FUNCTION_BLOCK FB_MadgwickFilter
VAR_INPUT
    stAccelData : ST_3D_values; // Acceleration Data in (g)
    stGyroData : ST_3D_values; // Gyroscope Data in (°/s)
    fBeta: REAL := 0.05; // Algorithm gain
    fCycletime: REAL; // Time step (s)
    bSetReference: BOOL; // Flag to set reference position
END_VAR

VAR_OUTPUT
	fQ0 : LREAL := 1.0; // Quaternion component
    fQ1 : LREAL := 0.0; // Quaternion component
    fQ2 : LREAL := 0.0; // Quaternion component
    fQ3 : LREAL := 0.0; // Quaternion component
    stEulerAngle_deg : ST_3D_values; // Estimated Euler angle in degrees X= Pitch, Y=Roll, Z=Yaw
    stEulerAngle_rad : ST_3D_values; // Estimated Euler angle in rad X= Pitch, Y=Roll, Z=Yaw
END_VAR

VAR

	// Reference angles
	stRef_Angles_deg :ST_3d_values; // Reference orientation (bSetReference; angles in degrees)
    fNorm : LREAL;
    _2fQ0, _2fQ1, _2fQ2, _2fQ3 : LREAL;
    _4fQ0, _4fQ1, _4fQ2, _4fQ3 : LREAL;
    _8fQ1, _8fQ2 : LREAL;
    fQ0fQ0, fQ1fQ1, fQ2fQ2, fQ3fQ3 : LREAL;
    fAx, fAy, fAz : LREAL;
    fS1, fS2, fS3, fS4 : LREAL;
    fSinRoll, fCosRoll : LREAL;
    fSinPitch, fCosPitch : LREAL;
    fSinYaw, fCosYaw : LREAL;
	fGyroRateX_rad,fGyroRateY_rad, fGyroRateZ_rad:LREAL;
END_VAR

// Normalize accelerometer measurements
fAx := REAL_TO_LREAL(stAccelData.x);
fAy := REAL_TO_LREAL(stAccelData.y);
fAz := REAL_TO_LREAL(stAccelData.z);
fNorm := fAx * fAx + fAy * fAy + fAz * fAz;
IF fNorm > 1E-6 THEN
    fNorm := SQRT(fNorm);
    fAx := fAx / fNorm;
    fAy := fAy / fNorm;
    fAz := fAz / fNorm;
END_IF

// Estimated direction of gravity and magnetic field
_2fQ0 := 2.0 * fQ0;
_2fQ1 := 2.0 * fQ1;
_2fQ2 := 2.0 * fQ2;
_2fQ3 := 2.0 * fQ3;
_4fQ0 := 4.0 * fQ0;
_4fQ1 := 4.0 * fQ1;
_4fQ2 := 4.0 * fQ2;
_4fQ3 := 4.0 * fQ3;
_8fQ1 := 8.0 * fQ1;
_8fQ2 := 8.0 * fQ2;
fQ0fQ0 := fQ0 * fQ0;
fQ1fQ1 := fQ1 * fQ1;
fQ2fQ2 := fQ2 * fQ2;
fQ3fQ3 := fQ3 * fQ3;

// Gradient descent algorithm corrective step
fS1 := _4fQ0 * fQ2fQ2 + _2fQ2 * fAx + _4fQ0 * fQ1fQ1 - _2fQ1 * fAy;
fS2 := _4fQ1 * fQ3fQ3 - _2fQ3 * fAx + 4.0 * fQ0fQ0 * fQ1 - _2fQ0 * fAy - _4fQ1 + _8fQ1 * fQ1fQ1 + _8fQ1 * fQ2fQ2 + _4fQ1 * fAz;
fS3 := 4.0 * fQ0fQ0 * fQ2 + _2fQ0 * fAx + _4fQ2 * fQ3fQ3 - _2fQ3 * fAy - _4fQ2 + _8fQ2 * fQ1fQ1 + _8fQ2 * fQ2fQ2 + _4fQ2 * fAz;
fS4 := 4.0 * fQ1fQ1 * fQ3 - _2fQ1 * fAx + 4.0 * fQ2fQ2 * fQ3 - _2fQ2 * fAy;

// Normalize step magnitude
fNorm := fS1 * fS1 + fS2 * fS2 + fS3 * fS3 + fS4 * fS4;
IF fNorm > 1E-6 THEN
    fNorm := SQRT(fNorm);
    fS1 := fS1 / fNorm;
    fS2 := fS2 / fNorm;
    fS3 := fS3 / fNorm;
    fS4 := fS4 / fNorm;
END_IF

// Apply gradient descent corrective step
fQ0 := fQ0 - REAL_TO_LREAL(fBeta) * fS1 * REAL_TO_LREAL(fCycleTime);
fQ1 := fQ1 - REAL_TO_LREAL(fBeta) * fS2 * REAL_TO_LREAL(fCycleTime);
fQ2 := fQ2 - REAL_TO_LREAL(fBeta) * fS3 * REAL_TO_LREAL(fCycleTime);
fQ3 := fQ3 - REAL_TO_LREAL(fBeta) * fS4 * REAL_TO_LREAL(fCycleTime);

// Convert gyroscope rates from °/s to rad/s
fGyroRateX_rad := stGyroData.x * pi / 180.0;
fGyroRateY_rad := stGyroData.y * pi / 180.0;
fGyroRateZ_rad := stGyroData.z * pi / 180.0;

// Integrate rate of change of quaternion
fQ0 := fQ0 + 0.5 * (-fQ1 * REAL_TO_LREAL(fGyroRateX_rad) - fQ2 * REAL_TO_LREAL(fGyroRateY_rad) - fQ3 * REAL_TO_LREAL(fGyroRateZ_rad)) * REAL_TO_LREAL(fCycleTime);
fQ1 := fQ1 + 0.5 * (fQ0 * REAL_TO_LREAL(fGyroRateX_rad) + fQ2 * REAL_TO_LREAL(fGyroRateZ_rad) - fQ3 * REAL_TO_LREAL(fGyroRateY_rad)) * REAL_TO_LREAL(fCycleTime);
fQ2 := fQ2 + 0.5 * (fQ0 * REAL_TO_LREAL(fGyroRateY_rad) - fQ1 * REAL_TO_LREAL(fGyroRateZ_rad) + fQ3 * REAL_TO_LREAL(fGyroRateX_rad)) * REAL_TO_LREAL(fCycleTime);
fQ3 := fQ3 + 0.5 * (fQ0 * REAL_TO_LREAL(fGyroRateZ_rad) + fQ1 * REAL_TO_LREAL(fGyroRateY_rad) - fQ2 * REAL_TO_LREAL(fGyroRateX_rad)) * REAL_TO_LREAL(fCycleTime);

// Normalize quaternion
fNorm := fQ0 * fQ0 + fQ1 * fQ1 + fQ2 * fQ2 + fQ3 * fQ3;
IF fNorm > 1E-6 THEN
    fNorm := SQRT(fNorm);
    fQ0 := fQ0 / fNorm;
    fQ1 := fQ1 / fNorm;
    fQ2 := fQ2 / fNorm;
    fQ3 := fQ3 / fNorm;
END_IF

// Calculate trigonometric values directly from quaternion components
fSinRoll := 2.0 * (fQ0 * fQ1 + fQ2 * fQ3);
fCosRoll := 1.0 - 2.0 * (fQ1 * fQ1 + fQ2 * fQ2);
fSinPitch := 2.0 * (fQ0 * fQ2 - fQ3 * fQ1);
fCosPitch := 1.0 - 2.0 * (fQ2 * fQ2 + fQ3 * fQ3);
fSinYaw := 2.0 * (fQ0 * fQ3 + fQ1 * fQ2);
fCosYaw := 1.0 - 2.0 * (fQ3 * fQ3 + fQ2 * fQ2);

// Convert trigonometric values to Euler angles using ATAN2 and ASIN in radians
stEulerAngle_rad.y := LREAL_TO_REAL(ATAN2(fSinRoll, fCosRoll));
stEulerAngle_rad.x := LREAL_TO_REAL(ASIN(fSinPitch));
stEulerAngle_rad.Z := LREAL_TO_REAL(ATAN2(fSinYaw, fCosYaw));

// Convert radians to degrees
stEulerAngle_deg.y := stEulerAngle_rad.y * 180.0 / pi;
stEulerAngle_deg.x := stEulerAngle_rad.x * 180.0 / pi;
stEulerAngle_deg.z := stEulerAngle_rad.z * 180.0 / pi;

// Set reference position if flag is active
IF bSetReference THEN
    stRef_Angles_deg.X := stEulerAngle_deg.X;
    stRef_Angles_deg.Y := stEulerAngle_deg.Y;
    stRef_Angles_deg.Z := stEulerAngle_deg.Z;
END_IF

// Apply reference position
stEulerAngle_deg.X := stEulerAngle_deg.X - (stRef_Angles_deg.X);
stEulerAngle_deg.Y := stEulerAngle_deg.Y - (stRef_Angles_deg.Y);
stEulerAngle_deg.Z := stEulerAngle_deg.Z - (stRef_Angles_deg.Z);

stEulerAngle_rad.X := stEulerAngle_rad.X - (stRef_Angles_deg.X) * PI / 180.0;
stEulerAngle_rad.Y := stEulerAngle_rad.Y - (stRef_Angles_deg.Y) * PI / 180.0;
stEulerAngle_rad.Z := stEulerAngle_rad.Z - (stRef_Angles_deg.Z) * PI / 180.0;

END_FUNCTION_BLOCK

(* stored: Version 1.1.0.1, ProductVersion 3.1.4024.13
   POU FB_MadgwickFilter: Id {c39968fe-236e-4aec-8c66-b5458e598e13}, SpecialFunc None *)
